PROGRAM S10_BeltCarrying
VAR
	//工站
	station					: REFERENCE TO FB_Station:=fbstation[10];
	//气缸
	
	//伺服
	fbROTAxisMove	 :REFERENCE TO FB_Axis:=fbAxis[16];	//	出料线体伺服
	
	//延时
	arTonDelay :ARRAY[1..20] OF TON;
	//返回值
	UdiReturnValue :ARRAY[1..20] OF UDINT;
	//过程记录
	tsModuleProcess:ARRAY[1..gc_ModuleProNo] OF DUT_Process;
	xClearModuleProcessDone:BOOL;
	bClearProcessStep	:BYTE;
	i,t: INT;
	bCounter:BYTE;

	 //报警屏蔽
	_AlarmDisable: BOOL;
	//首次循环
	_FirstCycle: ARRAY[1..10]OF BOOL;
	// //入料允许
	xBeltMovingEnable: BOOL;
	wActionCalibration: WORD;
	// 起始位置
	rStartPoition: ARRAY[0..8] OF REAL;
	// 结束位置
	rEndPoition:ARRAY[0..8] OF  REAL;
	NextPosR_TRIG: R_TRIG;
	tes: REAL;
	// 深孔板检测传感器
	xBoxSensorReached: ARRAY[1..2] of BOOL;
	xNotStop: BOOL;
	// 间距
	rcalcPos: ARRAY[0..7] OF REAL;
	//平均数
	raverage:REAL;
	_xFirstCycle: BOOL;
END_VAR

A_Input();
Alarm();
Delay();
FlowAuto();
FlowInit();
General();
ILC();
TipAuto();
TipManual();
Z_Output();

ACTION A_Input:
//气缸
//传感器
xBoxSensorReached[1]:=IxBeltEntryBoxCheckSensor2	;//	皮带线入口处¶深孔板检测传感器1
xBoxSensorReached[2]:=IxBeltEntryBoxCheckSensor1	;//	皮带线入口处¶深孔板检测传感器2

//允许进料
xBeltMovingEnable:=sModbus_200SMART.iBeltEnterEnable =1;
END_ACTION

ACTION Alarm:
//
station.adwAlarm[1].00:=station.xInitTimeout;	  			//S09CardCarrying 初始化超时
END_ACTION

ACTION Delay:
arTonDelay[01](IN:= , PT:=T#0.1S , Q=> , ET=> );
(*arTonDelay[02](IN:=  , PT:=T#1S , Q=> , ET=> );*)//已被使用
(*arTonDelay[03](IN:=   , PT:=T#1S , Q=> , ET=> );*)//已被使用
arTonDelay[04](IN:= , PT:=T#0.1S , Q=> , ET=> );
arTonDelay[05](IN:= , PT:=T#0.1S , Q=> , ET=> );
arTonDelay[06](IN:= , PT:=T#0.1S , Q=> , ET=> );
arTonDelay[07](IN:= , PT:=T#0.1S , Q=> , ET=> );
arTonDelay[08](IN:= , PT:=T#0.1S , Q=> , ET=> );
arTonDelay[09](IN:= , PT:=T#0.1S , Q=> , ET=> );
arTonDelay[10](IN:= NOT fbROTAxisMove.xbusy , PT:=T#0.1S , Q=> , ET=> );//TipAuto使用
END_ACTION

ACTION FlowAuto:

//-----------------------------------------初始化是否完成判断----------------------------------------------
IF NOT station.xInitDone 
THEN
 	station.iStepAuto:=0;
 	station.xDone:=FALSE;
ELSIF station.xRunning   OR 
(tsModuleProcess[1].xProcessStarted AND NOT tsModuleProcess[1].xProcessCompleted) OR//皮带线伺服移动
(tsModuleProcess[2].xProcessStarted AND NOT tsModuleProcess[2].xProcessCompleted)  //皮带线回原点
THEN
//-----------------------------------------动作步骤--------------------------------------------------------
CASE station.iStepAuto OF	  
	0: //----Home Step，等待启动----
		IF station.xDisabled 
			AND station.xCanRun 
			AND NOT fbMachine[1].xStopped 
			AND NOT station.xSingleRunning 
		THEN
			station.xDone:=TRUE;
		END_IF
		
		IF  station.xSingleRunning 
			OR station.xCanRun 
			//AND NOT station.xDone 
			AND NOT station.xDisabled 
			AND NOT fbMachine[1].xStopped
		THEN
			station.xCycleEnable:=TRUE;
			//station.xDone:= FALSE;  
			
			station.iStepAuto:= 10;
		END_IF
    10: //复位数据 
			IF  station.xSingleRunning THEN
				 FOR i:=1 TO gc_ModuleProNo BY 1 DO
						 MEMSET(ADR(tsModuleProcess[i]),0,SIZEOF(tsModuleProcess[i]));
				 END_FOR
			END_IF
			station.iStepAuto:=15;
	15://等待工位完成信号
		IF  NOT  fbMachine[1].xTryRun AND   NOT station.xSingleRunning THEN 
			IF  S07_BoxCarrying.station.xDone  AND 
				S09_CardCarrying.station.xDone  AND (xBeltMovingEnable OR S11_Packing.station.xDisabled ) THEN
					station.iStepAuto:=25;
			END_IF
		ELSE
		 			station.iStepAuto:=25;
		END_IF
	25://不允许各工位放料
				station.xDone :=FALSE;
				station.iStepAuto:=80;	   
	80://
				tsModuleProcess[1].xProcessNotStarted:=TRUE;
			  rStartPoition[t]:=fbROTAxisMove.rActPos;
				station.iStepAuto:=90;
	90://储存当前位置
			stData.Axis[16].rMovePosition[3]:=fbROTAxisMove.rActPos;
			station.iStepAuto:=95;
	95://读取原点偏移量
		 IF NOT _xFirstCycle THEN
		   stData.Axis[16].rMovePosition[2] := stData.Axis[16].rMovePosition[1] ;
		   _xFirstCycle := TRUE ;
		 END_IF
		   station.iStepAuto:=110;	
	//100://判断伺服位置是否合理
	//		IF      ( ABS(stData.Axis[16].rMovePosition[3]+stData.Axis[16].rRelativeDistance))+0.1>=ABS(stData.Axis[16].rMovePosition[2]) AND 
	//				  ( ABS(stData.Axis[16].rMovePosition[3]+stData.Axis[16].rRelativeDistance))-0.1<=ABS(stData.Axis[16].rMovePosition[2]) THEN
	//				  station.iStepAuto:=120;(*伺服已经移动过了*)
	//		ELSIF  ABS(stData.Axis[16].rMovePosition[3])+0.1>=ABS(stData.Axis[16].rMovePosition[2]) AND 
	//			   ABS(stData.Axis[16].rMovePosition[3])-0.1<=ABS(stData.Axis[16].rMovePosition[2]) THEN
	//			     station.iStepAuto:=110;(*伺服需要移动*)
	//		END_IF
	110://数据更新 位置
				 tsModuleProcess[1].xProcessStarted:=TRUE;
				 stData.Axis[16].rMovePosition[2] := stData.Axis[16].rMovePosition[2] +stData.Axis[16].rRelativeDistance ;
				 arTonDelay[03](IN:= FALSE , PT:=T#50MS , Q=> , ET=> );
				 station.iStepAuto:= 120;
	120:
					arTonDelay[03](IN:= TRUE , PT:=T#50MS , Q=> , ET=> );
					IF arTonDelay[03].Q THEN
						 station.iStepAuto:=130;
				 			arTonDelay[03](IN:=FALSE, PT:=T#50MS , Q=> , ET=> );
				   END_IF
	130:
					fbROTAxisMove.xMoveAuto[2]:=TRUE;
				 IF fbROTAxisMove.xMoveInPos[2] THEN
					 station.iStepAuto :=140; 
				 END_IF	
	140://计算链条移动次数
				tsModuleProcess[1].xProcessCompleted:=TRUE;
				bCounter:=bCounter +1;
				station.iStepAuto:=142;	
	142://是否需要回原点
			  IF 	bCounter >8 THEN
						station.iStepAuto:=1000;	
				ELSE
				 			station.iStepAuto:=150;	
				END_IF
	150://数据传递
			FOR i:=4 TO 1 BY -1 DO
						MEMCPY(ADR(arBeltLineFixtureData[i+2]),ADR(arBeltLineFixtureData[i]),SIZEOF(arBeltLineFixtureData[i]));
			END_FOR
			 station.iStepAuto:=160;
	160://启动各个工位
			fbStation[7].xDone:=FALSE;
			fbStation[9].xDone:=FALSE;
			station.iStepAuto:=500;	
	500://清除本站过程记录
			FOR i:=1 TO gc_ModuleProNo BY 1 DO
				MEMSET(ADR(tsModuleProcess[i]),0,SIZEOF(tsModuleProcess[i]));
			END_FOR
			 station.iStepAuto:=999;
			
	999://----Single Run Finish----
		station.iStepAuto :=0;
		IF NOT station.xSingleContinuousRun THEN
			station.xSingleRunFlag:=FALSE;
		END_IF
		station.xCycleEnable:=FALSE;	
		station.xDone:=TRUE;	

1000://回原点流程
				fbROTAxisMove.xReferenceAuto := TRUE ;
				station.iStepAuto:=1010;	
1010://伺服回原点完成
	IF  fbAxisHome[16].home_done THEN 
		 fbROTAxisMove.xReferenceAuto  := FALSE ;
		 	station.iStepAuto:=1050;	
	END_IF
//1020://如果有报警
//		IF		fbROTAxisMove.xError THEN
//		 		fbROTAxisMove.xAlarmResetHmi:=TRUE;
//		ELSE
//		 		fbROTAxisMove.xAlarmResetHmi:=FALSE;	
//				 station.iStepAuto:=1050;	  
//		END_IF
1050://回原点完成
				tsModuleProcess[2].xProcessCompleted:=TRUE;
				_xFirstCycle:=FALSE;
				bCounter:=1;	
				station.iStepAuto:=142;	
				


	
	ELSE
		;	
END_CASE
END_IF
END_ACTION

ACTION FlowInit:
IF NOT station.xIniting THEN
  station.iStepInit:=0;    
ELSE
//--------------------------------------------初始化步序----------------------------------
CASE station.iStepInit OF	
 0://  
  	IF station.xIniting THEN	
  	  station.iStepInit:=10;	
  	END_IF	
10://复位数据
	bCounter:=1;
	_xFirstCycle:=FALSE;
	station.iStepInit:=20;
20://伺服上电
	fbROTAxisMove.xPowerInit :=TRUE;
	IF  fbROTAxisMove.xPowerOn THEN
			station.iStepInit:=30;
	END_IF
30: //伺服回原点
	fbROTAxisMove.xReferenceAuto := TRUE ;
	station.iStepInit:=40;
40://伺服回原点完成
	IF  fbAxisHome[16].home_done THEN 
		 fbROTAxisMove.xReferenceAuto  := FALSE ;
		 station.iStepInit:=50;  
	END_IF
50: //再次伺服回原点，保证位置
	fbROTAxisMove.xReferenceAuto := TRUE ;
	station.iStepInit:=60;
60://伺服回原点完成
	IF  fbAxisHome[16].home_done THEN 
		 fbROTAxisMove.xReferenceAuto  := FALSE ;
		 station.iStepInit:=70;  
	END_IF	
//65://如果有报警
//		IF		fbROTAxisMove.xError THEN
//		 		fbROTAxisMove.xAlarmResetHmi:=TRUE;
//		ELSE
//		 		fbROTAxisMove.xAlarmResetHmi:=FALSE;	
//				 station.iStepInit:=70;  
//		END_IF
70://伺服去待机点
	fbROTAxisMove.xMoveAuto[1]:=TRUE;
	IF  fbROTAxisMove.xMoveInPos[1] THEN
		 station.iStepInit:=999; 
	END_IF
999://初始化完成	
	station.iStepInit:=0;
	station.xInitDone:=TRUE;  
END_CASE
END_IF
END_ACTION

ACTION General:
{region "计算环形线周长程序"}
CASE wActionCalibration OF   
  10://回原点
  fbROTAxisMove.xReferenceAuto:= TRUE ;
  	wActionCalibration:=15;
  15:
	 IF  fbAxisHome[16].home_done THEN 
		 fbROTAxisMove.xReferenceAuto  := FALSE ;
		wActionCalibration:=100;
	 END_IF
  20://Jog正向，遇到原点传感器停止
   stData.Axis[16].rJogVelocity :=0.1;  
	fbROTAxisMove.xJogForwardAuto := TRUE ;
	 IF  arAxisSensorH[16] THEN 
		 fbROTAxisMove.xJogForwardAuto := FALSE ; 
			wActionCalibration:=30;
			rStartPoition[t]:=fbROTAxisMove.rActPos;
	 END_IF 
  60: //高速走定位，理论值前10MM处停止
	stData.Axis[16].rMovePosition[5] :=(755*5)-10; 
	wActionCalibration:=70;
	
70:
	fbROTAxisMove.xMoveAuto[5] := TRUE ;
	 IF fbROTAxisMove.xMoveInPos[5] THEN 
	 fbROTAxisMove.xMoveAuto[5] := FALSE ; 
	 wActionCalibration:=80;
	 END_IF 
80:
	  stData.Axis[16].rJogVelocity :=0.1;  
	fbROTAxisMove.xJogForwardAuto := TRUE ;
 IF   arAxisSensorH[16] THEN 
	 fbROTAxisMove.xJogForwardAuto := FALSE ; 
 		wActionCalibration:=90;
		rEndPoition[t]:=fbROTAxisMove.rActPos;
 END_IF 
90:
		stData.Axis[16].rRelativeDistance:=((rEndPoition[t]-rStartPoition[t])/85);
		wActionCalibration:=0;
END_CASE  
  
{endregion}
	 
{region "去下一个位置"}
NextPosR_TRIG(CLK:= fbMachine[1].xManualMode AND fbROTAxisMove.xMoveHmi[6], Q=> );
IF  NextPosR_TRIG.Q THEN
 stData.Axis[16].rMovePosition[6]:=fbROTAxisMove.rActPos +fbROTAxisMove.rRelativeDistance;
END_IF
  
{endregion}
END_ACTION

ACTION ILC:

//---------------------------------------------------工站可执行-------------------------------------------------------
station.xCanRun :=TRUE ;

//---------------------------------------------------气缸动作条件-------------------------------------------



//---------------------------------------------------伺服动作条件-------------------------------------------



fbROTAxisMove.xRunILC := 
fbROTAxisMove.xMoveILC[1] :=
fbROTAxisMove.xMoveILC[2] :=
fbROTAxisMove.xMoveILC[3] :=
fbROTAxisMove.xMoveILC[4] :=
fbROTAxisMove.xMoveILC[5] := TRUE ;
fbROTAxisMove.xRelativeILC:=TRUE;
END_ACTION

ACTION TipAuto:

//------------------------------------------------AutoTip Cylinder--------------------------------
//------------------------------------------------AutoTip Servo--------------------------------
//**************************************
//FOR i:= 1 TO 5 BY 1 DO 
//	IF fbROTAxisMove.xMoveAuto[i] THEN
//		fbROTAxisMove.iPosNumber := i ;
//	END_IF
//	
//END_FOR
//
//
//IF  fbMachine[1].xAutoMode AND NOT fbMachine[1].xRunning AND arTonDelay[10].Q   THEN
//	IF	fbROTAxisMove.iPosNumber=1 	AND NOT fbROTAxisMove.xMoveInPos[1] 	THEN 	station.adwAutoTip[1].10:=TRUE	;	END_IF//轴伺服自动时位置不在位置1
//	if	fbROTAxisMove.iPosNumber=2	AND NOT fbROTAxisMove.xMoveInPos[2]	THEN 	station.adwAutoTip[1].11:=TRUE	;	END_IF//轴伺服自动时位置不在位置2
//	if	fbROTAxisMove.iPosNumber=3	AND NOT fbROTAxisMove.xMoveInPos[3]	THEN 	station.adwAutoTip[1].12:=TRUE	;	END_IF//轴伺服自动时位置不在位置3
//	if	fbROTAxisMove.iPosNumber=4	AND NOT fbROTAxisMove.xMoveInPos[4]	THEN 	station.adwAutoTip[1].13:=TRUE	;	END_IF//轴伺服自动时位置不在位置4
//	IF	fbROTAxisMove.iPosNumber=5	AND NOT fbROTAxisMove.xMoveInPos[5]	THEN 	station.adwAutoTip[1].14:=TRUE	;	END_IF//轴伺服自动时位置不在位置5
//END_IF
END_ACTION

ACTION TipManual:
//--------------------------------------------ManualTip------------------------------------------------------

//-------------------------------------------气缸提示---------------------------------------------------------




/////////////////////////////////////////////////////////////////////////////////////////////////////////////////
END_ACTION

ACTION Z_Output:
(**************************气缸输出********************************)
END_ACTION

END_PROGRAM

(* stored: Version 1.1.0.1, ProductVersion 3.1.4024.9
   POU S10_BeltCarrying: Id {f14c7987-78b0-43f4-9505-460a33d7d0cf}, SpecialFunc None
   Action A_Input: Id {5549612f-f835-4cac-8e2f-81ddd47e4429}
   Action Alarm: Id {f100fef2-7bd1-4fe4-a530-9448d1f71b42}
   Action Delay: Id {3e6d0638-113c-4b73-a71d-99982a90a940}
   Action FlowAuto: Id {150835d7-b6d9-4f7e-b17a-65598f78bf7a}
   Action FlowInit: Id {8c3c079e-1f18-47e9-9b8f-ac261d5376ea}
   Action General: Id {0cae7ce3-2c84-4098-b25b-44511bfb9f95}
   Action ILC: Id {92fad71f-f937-4458-b440-4469ed850f69}
   Action TipAuto: Id {7d0b378b-5f23-4601-b0e9-fba22d16cc5e}
   Action TipManual: Id {234546c3-9ee4-4897-926f-08de62e253ec}
   Action Z_Output: Id {580bf8d9-96ef-467f-a5e7-158e7bf5ab7c} *)
